# EPICS autosave request: req/motor_settings.req
$(P)$(M).DHLM
$(P)$(M).DLLM
$(P)$(M).VELO
$(P)$(M).VMAX
$(P)$(M).OFF
$(P)$(M).MRES
$(P)$(M).ERES
$(P)$(M).PREC
$(P)$(M).EGU
$(P)$(M).TWV
$(P)$(M).RDBD
